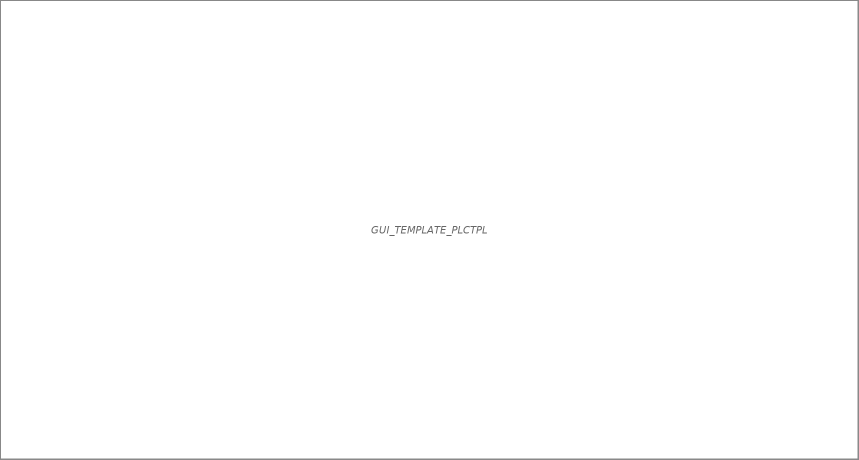
VISUALIZATION GUI_Device001  // 859x460
    Frame (0,0 859x460)
        shows GUI_TEMPLATE_PLCTPL(m_Instance := MAIN.Device001)
END_VISUALIZATION

(* stored: Version 1.1.0.1, ProductVersion 3.1.4024.3
   Visu GUI_Device001: Id {05fa3a21-cc3f-46e4-a133-64595b3fadfd} *)
